// TIA Portal V18 export
// export: Created 2026-06-20T23:26:23.319602Z, ExportSetting WithDefaults
TextList "TL_Phan_Quyen"  ListRange=Decimal, Comment="Phân quyền vận hành"
  TextListEntry   EntryType=SingleValue, Text="Chưa đăng nhập"
  TextListEntry   EntryType=SingleValue, From=1, To=1, Text="Operator - Start/Stop, Ack Alarm, xem màn hình"
  TextListEntry   EntryType=SingleValue, From=2, To=2, Text="Engineer - sửa thông số, manual, reset alarm"
  TextListEntry   EntryType=SingleValue, From=3, To=3, Text="Admin - toàn quyền"
